RESOURCE_TYPE _Core022
  (* Standard: 61499-2 *)
  (* Version 0.1, 2017-00-06, Hammond, HAMMONDSDESKTOP *)
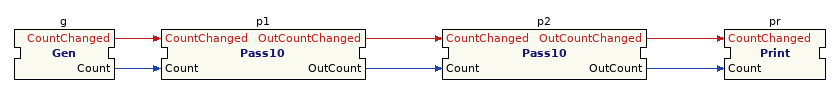
  FBS
    g : Gen;
    p1 : Pass10;
    p2 : Pass10;
    pr : Print;
  END_FBS
  EVENT_CONNECTIONS
    g.CountChanged TO p1.CountChanged;
    p1.OutCountChanged TO p2.CountChanged;
    p2.OutCountChanged TO pr.CountChanged;
  END_CONNECTIONS
  DATA_CONNECTIONS
    g.Count TO p1.Count;
    p1.OutCount TO p2.Count;
    p2.OutCount TO pr.Count;
  END_CONNECTIONS
END_RESOURCE_TYPE
